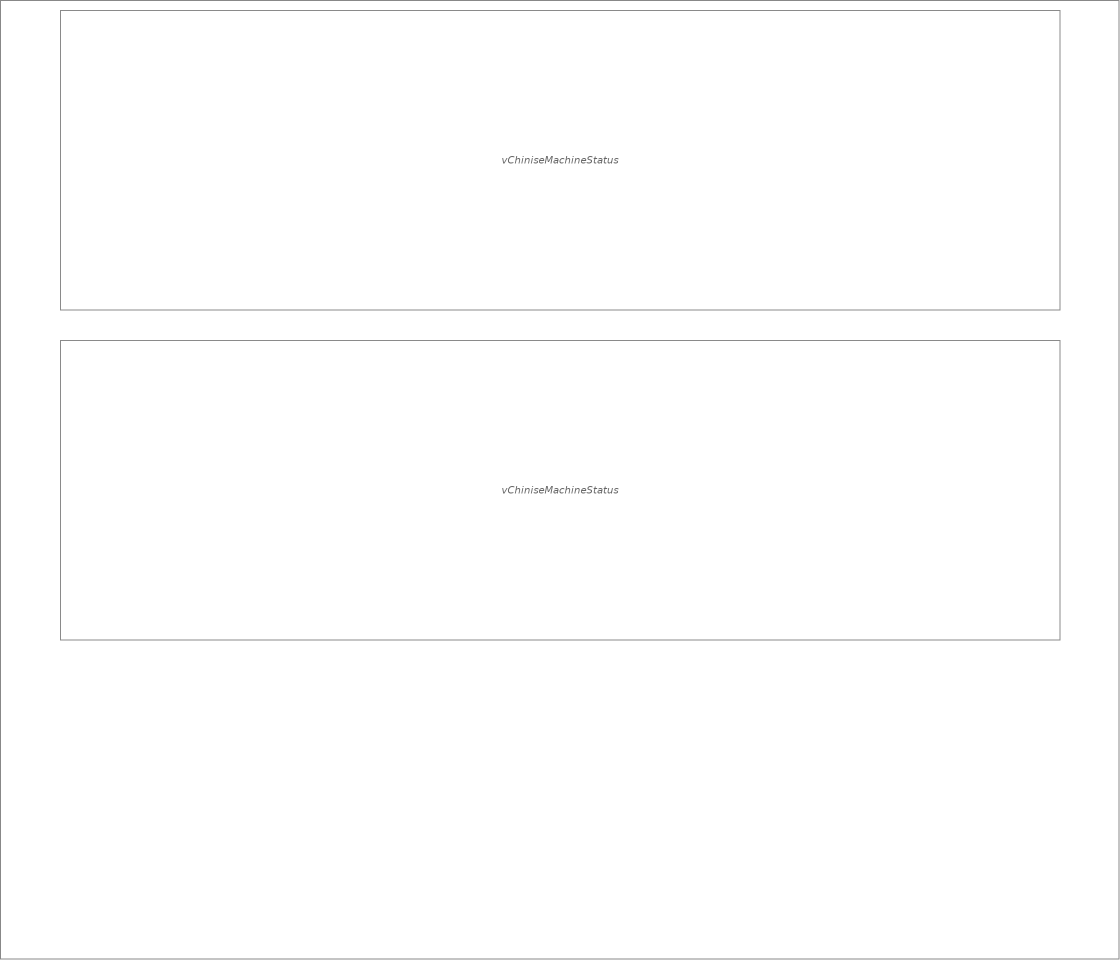
VISUALIZATION vFrameFillingLine_2  // 1120x960
VAR_IN_OUT

END_VAR
VAR
		iFiller_A 	: UINT := 0;
	iCork 		: UINT := 1;
	iFiller_B 	: UINT := 2;
	iSticker	: UINT := 3;
	iLaser		: UINT := 4;
END_VAR
    Frame (60,340 1000x300)
        shows vChiniseMachineStatus(stData := GVL.st_Laser_MachineSettings.stPimData, fbPIM := MAIN.fb_Laser_Station, iActualMachine := iLaser, fbModbusTCP := MAIN.fb_Laser_Machine.fbModbuCommunication, bTurnOnCommunication := GVL.st_Laser_MachineSettings.bCommunicationActive, iCommunicationCycleTime := GVL.st_Laser_MachineSettings.iCommunicationCycleTime)
    Frame (60,10 1000x300)
        shows vChiniseMachineStatus(stData := GVL.st_Sticker_MachineSettings.stPimData, fbPIM := MAIN.fb_Sticker_Station, iActualMachine := iSticker, fbModbusTCP := MAIN.fb_Sticker_Machine.fbModbuCommunication, bTurnOnCommunication := GVL.st_Sticker_MachineSettings.bCommunicationActive, iCommunicationCycleTime := GVL.st_Sticker_MachineSettings.iCommunicationCycleTime)
END_VISUALIZATION

(* stored: Version 1.1.0.1, ProductVersion 3.1.4024.13
   Visu vFrameFillingLine_2: Id {6f459862-92c6-47dc-b674-ea7537132465} *)
